% RSLogix 500 project project7.RSS, saved by version 8.30.00.16 %
PROJECT "UNTITLED"    % processor: Bul.1763 MicroLogix 1100 Series B %

PROGRAM FILES
  LAD 2 "MAIN"  4 rungs
  LAD 3 "IO"  3 rungs
  LAD 4 "CALIBRATE"  21 rungs
  LAD 5 "SAMPLE"  2 rungs

DATA FILES
  O0 OUTPUT  4 elements
  I1 INPUT  6 elements
  S2 STATUS  66 elements
  B3 BINARY  2 elements
  T4 TIMER  3 elements
  C5 COUNTER  1 elements
  R6 CONTROL  1 elements
  N7 INTEGER  10 elements
  F8 FLOAT  3 elements
  N9 INTEGER2  5 elements
  L10 LONG_INTEG  2 elements

LADDER 2 "MAIN"
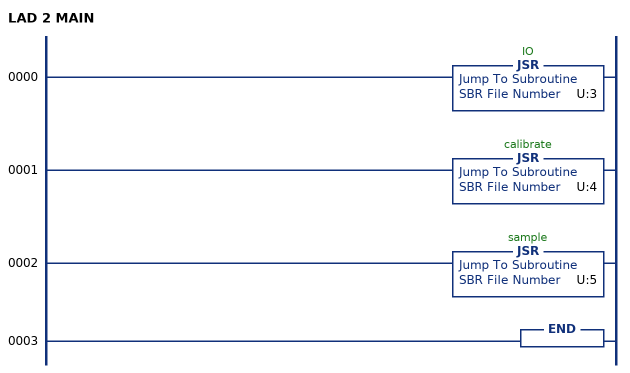
% Rung: 0 %
SOR JSR U:3 EOR
%   U:3  "IO" %
% Rung: 1 %
SOR JSR U:4 EOR
%   U:4  "calibrate" %
% Rung: 2 %
SOR JSR U:5 EOR
%   U:5  "sample" %
% Rung: 3 %
SOR END EOR

LADDER 3 "IO"
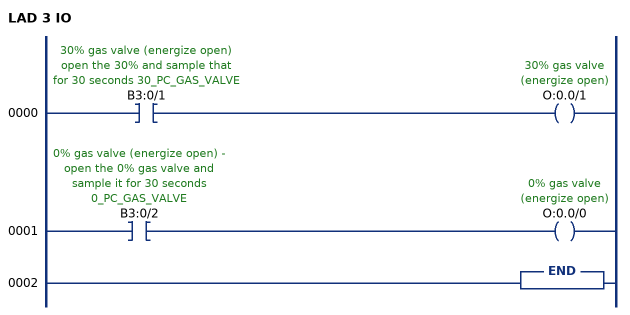
% Rung: 0 %
SOR XIC B3:0/1 OTE O:0.0/1 EOR
%   B3:0/1  30_PC_GAS_VALVE  "30% gas valve (energize open) open the 30% and sample that for 30 seconds" %
%   O:0.0/1  "30% gas valve (energize open)" %
% Rung: 1 %
SOR XIC B3:0/2 OTE O:0.0/0 EOR
%   B3:0/2  0_PC_GAS_VALVE  "0% gas valve (energize open) - open the 0% gas valve and sample it for 30 seconds" %
%   O:0.0/0  "0% gas valve (energize open)" %
% Rung: 2 %
SOR END EOR

LADDER 4 "CALIBRATE"
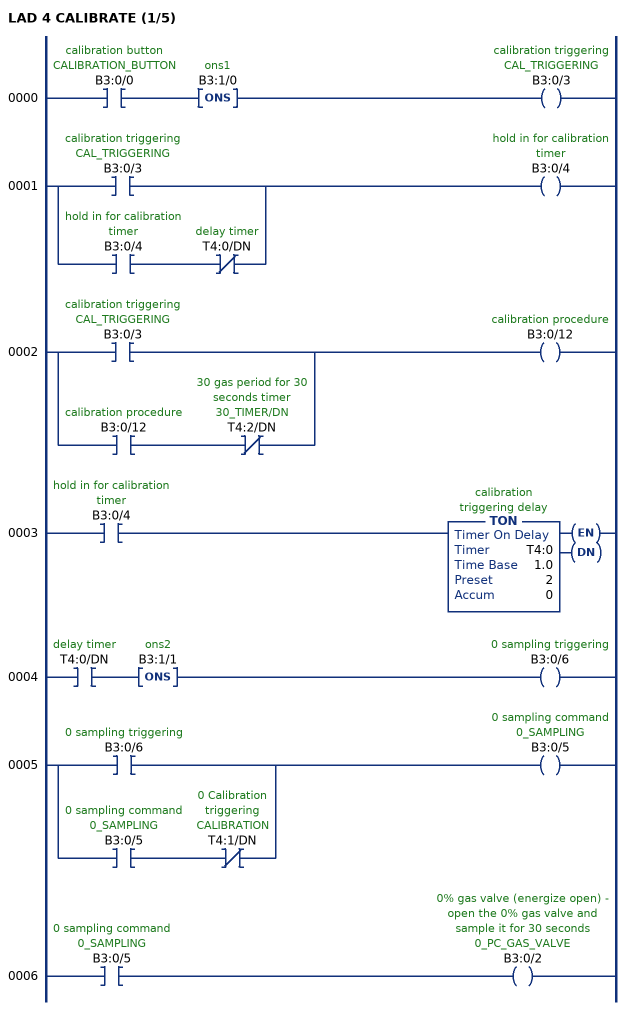
% Rung: 0 %
SOR XIC B3:0/0 ONS B3:1/0 OTE B3:0/3 EOR
%   B3:0/0  CALIBRATION_BUTTON  "calibration button" %
%   B3:1/0  "ons1" %
%   B3:0/3  CAL_TRIGGERING  "calibration triggering" %
% Rung: 1 %
SOR BST XIC B3:0/3 NXB XIC B3:0/4 XIO T4:0/DN BND OTE B3:0/4 EOR
%   B3:0/3  CAL_TRIGGERING  "calibration triggering" %
%   B3:0/4  "hold in for calibration timer" %
%   T4:0/DN  "delay timer" %
% Rung: 2 %
SOR BST XIC B3:0/3 NXB XIC B3:0/12 XIO T4:2/DN BND OTE B3:0/12 EOR
%   B3:0/3  CAL_TRIGGERING  "calibration triggering" %
%   B3:0/12  "calibration procedure" %
%   T4:2  30_TIMER  "30 gas period for 30 seconds timer" %
% Rung: 3 %
SOR XIC B3:0/4 TON T4:0 1.0 2 0 EOR
%   B3:0/4  "hold in for calibration timer" %
%   T4:0  "calibration triggering delay" %
% Rung: 4 %
SOR XIC T4:0/DN ONS B3:1/1 OTE B3:0/6 EOR
%   T4:0/DN  "delay timer" %
%   B3:1/1  "ons2" %
%   B3:0/6  "0 sampling triggering" %
% Rung: 5 %
SOR BST XIC B3:0/6 NXB XIC B3:0/5 XIO T4:1/DN BND OTE B3:0/5 EOR
%   B3:0/6  "0 sampling triggering" %
%   B3:0/5  0_SAMPLING  "0 sampling command" %
%   T4:1/DN  CALIBRATION  "0 Calibration triggering" %
% Rung: 6 %
SOR XIC B3:0/5 OTE B3:0/2 EOR
%   B3:0/5  0_SAMPLING  "0 sampling command" %
%   B3:0/2  0_PC_GAS_VALVE  "0% gas valve (energize open) - open the 0% gas valve and sample it for 30 seconds" %

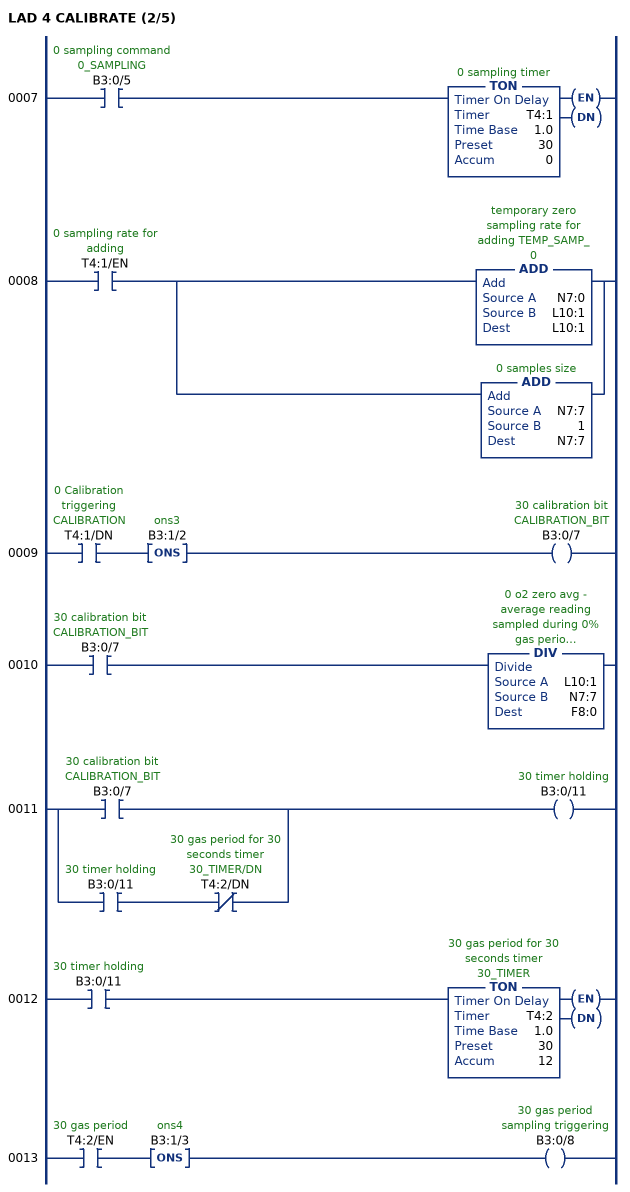
% Rung: 7 %
SOR XIC B3:0/5 TON T4:1 1.0 30 0 EOR
%   B3:0/5  0_SAMPLING  "0 sampling command" %
%   T4:1  "0 sampling timer" %
% Rung: 8 %
SOR XIC T4:1/EN BST ADD N7:0 L10:1 L10:1 NXB ADD N7:7 1 N7:7 BND EOR
%   T4:1/EN  "0 sampling rate for adding" %
%   N7:0  OXYGEN_INPUT  "O2 sensor input signal" %
%   L10:1  TEMP_SAMP_0  "temporary zero sampling rate for adding" %
%   N7:7  "0 samples size" %
% Rung: 9 %
SOR XIC T4:1/DN ONS B3:1/2 OTE B3:0/7 EOR
%   T4:1/DN  CALIBRATION  "0 Calibration triggering" %
%   B3:1/2  "ons3" %
%   B3:0/7  CALIBRATION_BIT  "30 calibration bit" %
% Rung: 10 %
SOR XIC B3:0/7 DIV L10:1 N7:7 F8:0 EOR
%   B3:0/7  CALIBRATION_BIT  "30 calibration bit" %
%   L10:1  TEMP_SAMP_0  "temporary zero sampling rate for adding" %
%   N7:7  "0 samples size" %
%   F8:0  O2_ZERO_AVERAGE_  "0 o2 zero avg - average reading sampled during 0% gas period" %
% Rung: 11 %
SOR BST XIC B3:0/7 NXB XIC B3:0/11 XIO T4:2/DN BND OTE B3:0/11 EOR
%   B3:0/7  CALIBRATION_BIT  "30 calibration bit" %
%   B3:0/11  "30 timer holding" %
%   T4:2  30_TIMER  "30 gas period for 30 seconds timer" %
% Rung: 12 %
SOR XIC B3:0/11 TON T4:2 1.0 30 12 EOR
%   B3:0/11  "30 timer holding" %
%   T4:2  30_TIMER  "30 gas period for 30 seconds timer" %
% Rung: 13 %
SOR XIC T4:2/EN ONS B3:1/3 OTE B3:0/8 EOR
%   T4:2/EN  "30 gas period" %
%   B3:1/3  "ons4" %
%   B3:0/8  "30 gas period sampling triggering" %

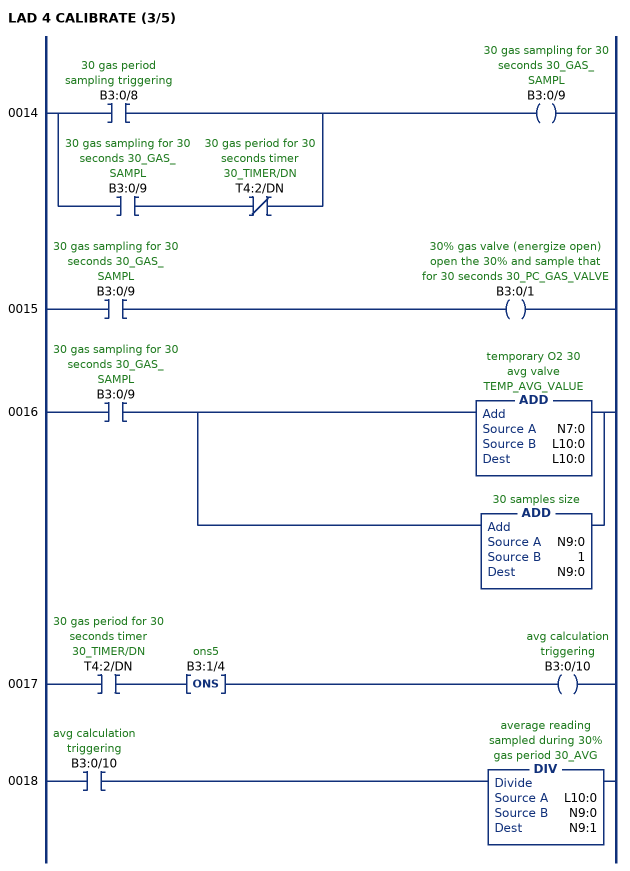
% Rung: 14 %
SOR BST XIC B3:0/8 NXB XIC B3:0/9 XIO T4:2/DN BND OTE B3:0/9 EOR
%   B3:0/8  "30 gas period sampling triggering" %
%   B3:0/9  30_GAS_SAMPL  "30 gas sampling for 30 seconds" %
%   T4:2  30_TIMER  "30 gas period for 30 seconds timer" %
% Rung: 15 %
SOR XIC B3:0/9 OTE B3:0/1 EOR
%   B3:0/9  30_GAS_SAMPL  "30 gas sampling for 30 seconds" %
%   B3:0/1  30_PC_GAS_VALVE  "30% gas valve (energize open) open the 30% and sample that for 30 seconds" %
% Rung: 16 %
SOR XIC B3:0/9 BST ADD N7:0 L10:0 L10:0 NXB ADD N9:0 1 N9:0 BND EOR
%   B3:0/9  30_GAS_SAMPL  "30 gas sampling for 30 seconds" %
%   N7:0  OXYGEN_INPUT  "O2 sensor input signal" %
%   L10:0  TEMP_AVG_VALUE  "temporary O2 30 avg valve" %
%   N9:0  "30 samples size" %
% Rung: 17 %
SOR XIC T4:2/DN ONS B3:1/4 OTE B3:0/10 EOR
%   T4:2  30_TIMER  "30 gas period for 30 seconds timer" %
%   B3:1/4  "ons5" %
%   B3:0/10  "avg calculation triggering" %
% Rung: 18 %
SOR XIC B3:0/10 DIV L10:0 N9:0 N9:1 EOR
%   B3:0/10  "avg calculation triggering" %
%   L10:0  TEMP_AVG_VALUE  "temporary O2 30 avg valve" %
%   N9:0  "30 samples size" %
%   N9:1  30_AVG  "average reading sampled during 30% gas period" %

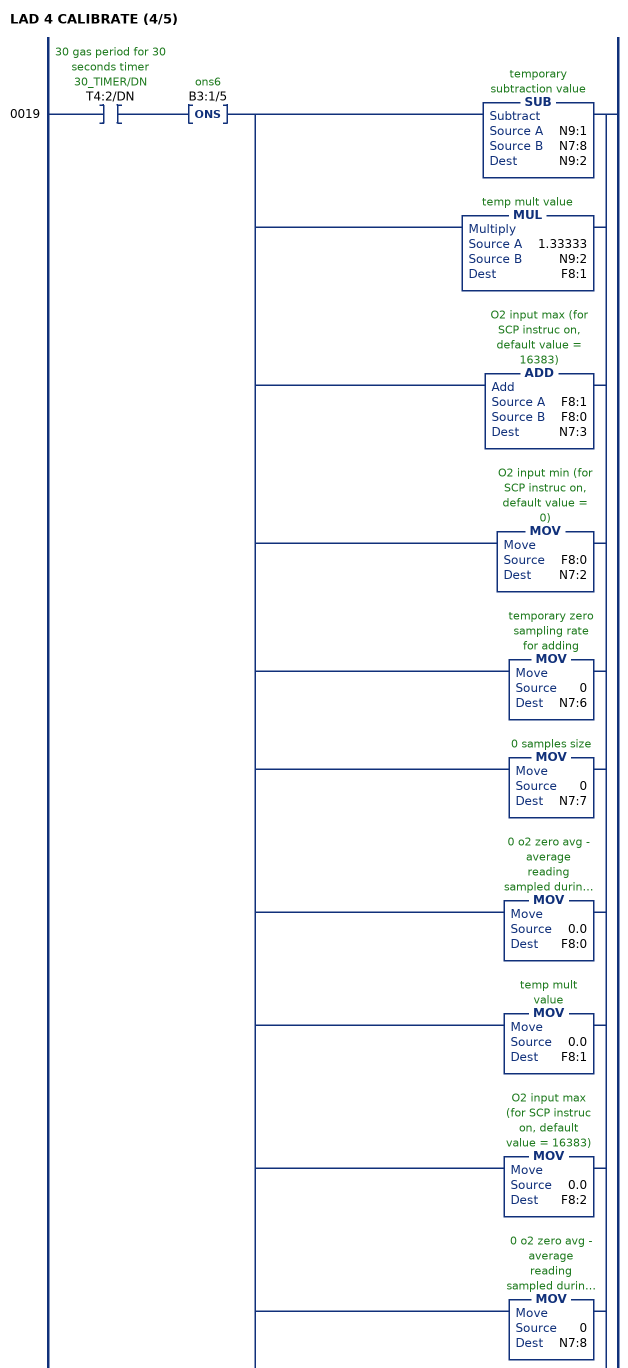

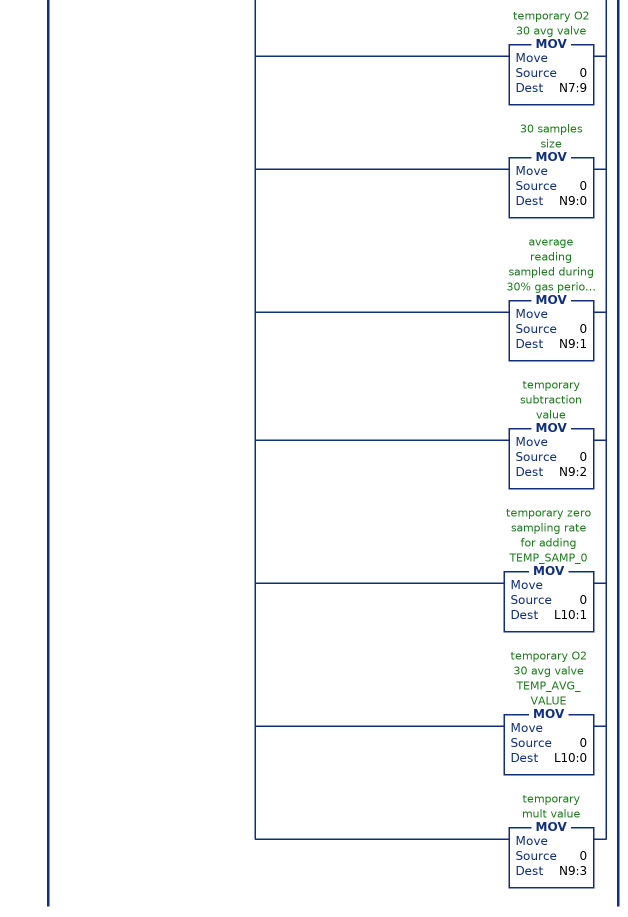
% Rung: 19 %
SOR XIC T4:2/DN ONS B3:1/5 BST SUB N9:1 N7:8 N9:2 NXB MUL 1.33333 N9:2 F8:1 NXB ADD F8:1 F8:0 N7:3 NXB MOV F8:0 N7:2 NXB MOV 0 N7:6 NXB MOV 0 N7:7 NXB MOV 0.0 F8:0 NXB MOV 0.0 F8:1 NXB MOV 0.0 F8:2 NXB MOV 0 N7:8 NXB MOV 0 N7:9 NXB MOV 0 N9:0 NXB MOV 0 N9:1 NXB MOV 0 N9:2 NXB MOV 0 L10:1 NXB MOV 0 L10:0 NXB MOV 0 N9:3 BND EOR
%   T4:2  30_TIMER  "30 gas period for 30 seconds timer" %
%   B3:1/5  "ons6" %
%   N9:1  30_AVG  "average reading sampled during 30% gas period" %
%   N7:8  O2_ZERO_AVERAGE  "0 o2 zero avg - average reading sampled during 0% gas period" %
%   N9:2  "temporary subtraction value" %
%   F8:1  "temp mult value" %
%   F8:0  O2_ZERO_AVERAGE_  "0 o2 zero avg - average reading sampled during 0% gas period" %
%   N7:3  "O2 input max (for SCP instruc on, default value = 16383)" %
%   N7:2  "O2 input min (for SCP instruc on, default value = 0)" %
%   N7:6  "temporary zero sampling rate for adding" %
%   N7:7  "0 samples size" %
%   F8:2  "O2 input max (for SCP instruc on, default value = 16383)" %
%   N7:9  "temporary O2 30 avg valve" %
%   N9:0  "30 samples size" %
%   L10:1  TEMP_SAMP_0  "temporary zero sampling rate for adding" %
%   L10:0  TEMP_AVG_VALUE  "temporary O2 30 avg valve" %
%   N9:3  "temporary mult value" %

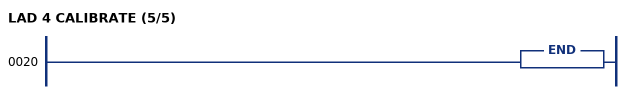
% Rung: 20 %
SOR END EOR

LADDER 5 "SAMPLE"
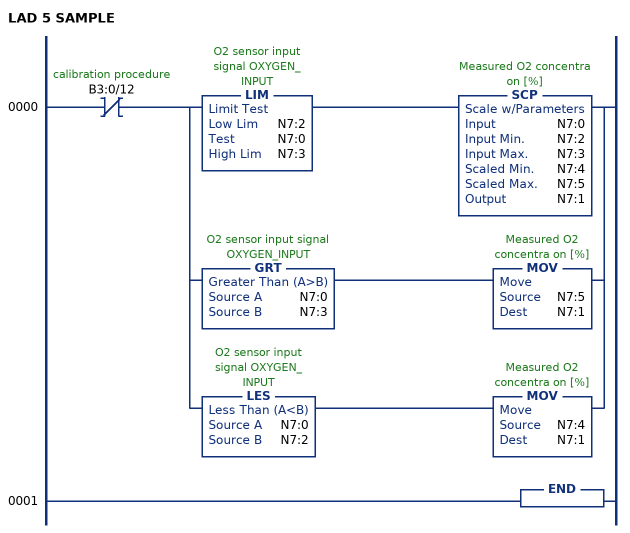
% Rung: 0 %
SOR XIO B3:0/12 BST LIM N7:2 N7:0 N7:3 SCP N7:0 N7:2 N7:3 N7:4 N7:5 N7:1 NXB GRT N7:0 N7:3 MOV N7:5 N7:1 NXB LES N7:0 N7:2 MOV N7:4 N7:1 BND EOR
%   B3:0/12  "calibration procedure" %
%   N7:2  "O2 input min (for SCP instruc on, default value = 0)" %
%   N7:0  OXYGEN_INPUT  "O2 sensor input signal" %
%   N7:3  "O2 input max (for SCP instruc on, default value = 16383)" %
%   N7:4  "lowest sensor range value" %
%   N7:5  "highest sensor range value" %
%   N7:1  "Measured O2 concentra on [%]" %
% Rung: 1 %
SOR END EOR

OTHER DOCUMENTED ADDRESSES
  N9:4  "4/3"

DATA TABLE (non-zero values as saved)
DATA T4
% .PRE .ACC %
% T4:0 % 2 0
% T4:1 % 30 0
% T4:2 % 30 12
DATA N7
% N7:0 % 0 0 0 16383 0 40 0 0 0 0
